TYPE (* A Structure with 16 BOOLS *)
  (* Version 1.0, 2024-02-21, franz *)
  ST16B : STRUCT
    B_00 : BOOL; (* BIT 00 *)
    B_01 : BOOL; (* BIT 01 *)
    B_02 : BOOL; (* BIT 02 *)
    B_03 : BOOL; (* BIT 03 *)
    B_04 : BOOL; (* BIT 04 *)
    B_05 : BOOL; (* BIT 05 *)
    B_06 : BOOL; (* BIT 06 *)
    B_07 : BOOL; (* BIT 07 *)
    B_08 : BOOL; (* BIT 08 *)
    B_09 : BOOL; (* BIT 09 *)
    B_10 : BOOL; (* BIT 10 *)
    B_11 : BOOL; (* BIT 11 *)
    B_12 : BOOL; (* BIT 12 *)
    B_13 : BOOL; (* BIT 13 *)
    B_14 : BOOL; (* BIT 14 *)
    B_15 : BOOL; (* BIT 15 *)
  END_STRUCT;
END_TYPE
